{attribute 'TcGenerated'}
{attribute 'no-analysis'}
{attribute 'linkalways'}
// This function has been automatically generated from the project information.
VAR_GLOBAL CONSTANT
	{attribute 'const_non_replaced'}
	stLibVersion_log4TC : ST_LibVersion := (iMajor := 0, iMinor := 2, iBuild := 3, iRevision := 0, nFlags := 0, sVersion := '0.2.3');
END_VAR

(* stored: Version 1.1.0.1, ProductVersion 3.1.4026.17
   GVL Global_Version: Id {7aeb1864-8588-48d9-bed3-fd1f47a849aa} *)
